{attribute 'pack_mode' := '1'}
TYPE ST_MoveAxisRelative EXTENDS ST_MsgToPLC:
STRUCT
    axisIndex	: DINT;
    distance	: LREAL;
    moveTime	: TIME;
END_STRUCT
END_TYPE

(* stored: Version 1.1.0.1, ProductVersion 3.1.4022.18
   DUT ST_MoveAxisRelative: Id {c2c2b5e6-c8e8-4cb0-8e05-7e03253b0949} *)
